{attribute 'enable_dynamic_creation'}
FUNCTION_BLOCK StepManagerBasic IMPLEMENTS IStepManager
VAR
    _currentStep : ENUM;
    _requestNumber : DINT;
END_VAR

// Copyright (c) 2024 Loupe (https://loupe.team), provided under the MIT License.

PROPERTY CurrentStepImpl : ENUM
GET
// Copyright (c) 2024 Loupe (https://loupe.team), provided under the MIT License.

CurrentStepImpl := _CurrentStep;
END_GET
END_PROPERTY

{warning 'add property implementation'}
PROPERTY RequestNumberImpl : DINT
GET
// Copyright (c) 2024 Loupe (https://loupe.team), provided under the MIT License.

RequestNumberImpl := _requestNumber;
END_GET
END_PROPERTY

METHOD RequestStepImpl : BOOL
VAR_INPUT
    nextStep : ENUM;
END_VAR
// Copyright (c) 2024 Loupe (https://loupe.team), provided under the MIT License.

_requestNumber := _requestNumber + 1;
_currentStep := nextStep;
END_METHOD

METHOD ResetImpl : BOOL
// Copyright (c) 2024 Loupe (https://loupe.team), provided under the MIT License.

_currentStep := SEQUENCE_STEP.NO_STEP;
END_METHOD

METHOD SequenceCompleteImpl : BOOL
// Copyright (c) 2024 Loupe (https://loupe.team), provided under the MIT License.

_requestNumber := _requestNumber + 1;
_currentStep := SEQUENCE_STEP.NO_STEP;
END_METHOD

METHOD SequenceErrorImpl : BOOL
VAR_INPUT
    ErrorCode : INT;
    ErrorMessage : STRING;
END_VAR
// Copyright (c) 2024 Loupe (https://loupe.team), provided under the MIT License.

_requestNumber := _requestNumber + 1;
_currentStep := SEQUENCE_STEP.NO_STEP;
END_METHOD

END_FUNCTION_BLOCK

(* stored: Version 1.1.0.1
   POU StepManagerBasic: Id {093266f8-f27d-447f-8d0c-4f60d6268941}, SpecialFunc None
   Property CurrentStepImpl: Id {29f4d86c-54a1-42a1-8dae-2fa8be71c206}
   Get Get: Id {6ff7d4db-2de2-41e3-931f-d828caaa0f1f}
   Property RequestNumberImpl: Id {56d18034-f9ba-490e-94ec-3c8b604cd6b0}
   Get Get: Id {3d104d88-59e8-4239-891c-6b40240640ee}
   Method RequestStepImpl: Id {631d6933-a3d4-4a04-8d8b-2defab756516}
   Method ResetImpl: Id {fb88c2f8-268f-48f3-8ad4-521cc35aeb3a}
   Method SequenceCompleteImpl: Id {ff6a8092-1516-4df4-b57d-1bb9d4d5c97b}
   Method SequenceErrorImpl: Id {a9f4d538-abc7-4246-9047-1ad6d24ed996} *)
